TYPE auxiliary_counters_code_enum :
(
	INFEED_REJECT_BARCODE				:= 1,
	INFEED_REJECT_HIGH_LOAD				:= 2,
	CROSSPUSHER_REJECT_LOW_LOAD			:= 3,
	CROSSPUSHER_REJECT_HIGH_LOAD		:= 4,
	CASE_FEED_REJECT					:= 5,
	TOTAL_UNITS							:= 7	
);
END_TYPE

(* stored: Version 1.1.0.1, ProductVersion 3.1.4024.3
   DUT auxiliary_counters_code_enum: Id {bfbc4f4a-046d-453f-b76e-cbe5aea27cc0} *)
